Xinje XCPPro project, PLC1: XC3-32 (software 3.3q 2016-08-30)

PROGRAM Ladder

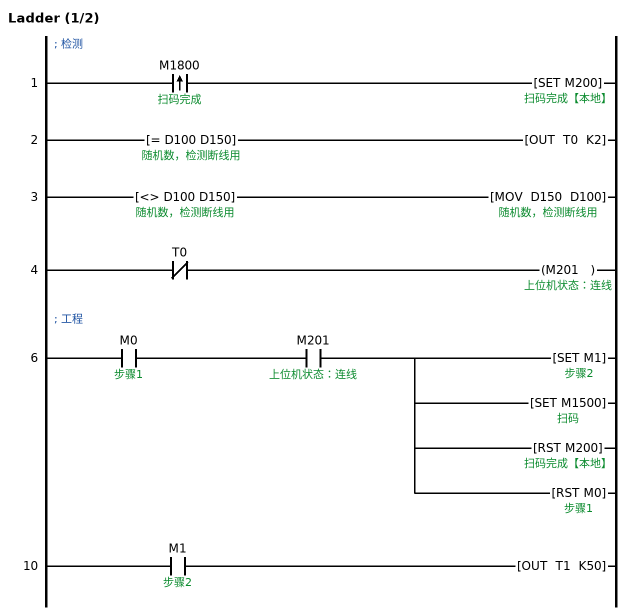
; 检测
LDP    M1800	; 扫码完成
SET    M200	; 扫码完成【本地】
LD=    D100 D150	; 随机数，检测断线用
OUT    T0 K2
LD<>   D100 D150	; 随机数，检测断线用
MOV    D150 D100	; 随机数，检测断线用
LDI    T0
OUT    M201	; 上位机状态：连线
; 工程
LD     M0	; 步骤1
AND    M201	; 上位机状态：连线
SET    M1	; 步骤2
SET    M1500	; 扫码
RST    M200	; 扫码完成【本地】
RST    M0	; 步骤1
LD     M1	; 步骤2
OUT    T1 K50

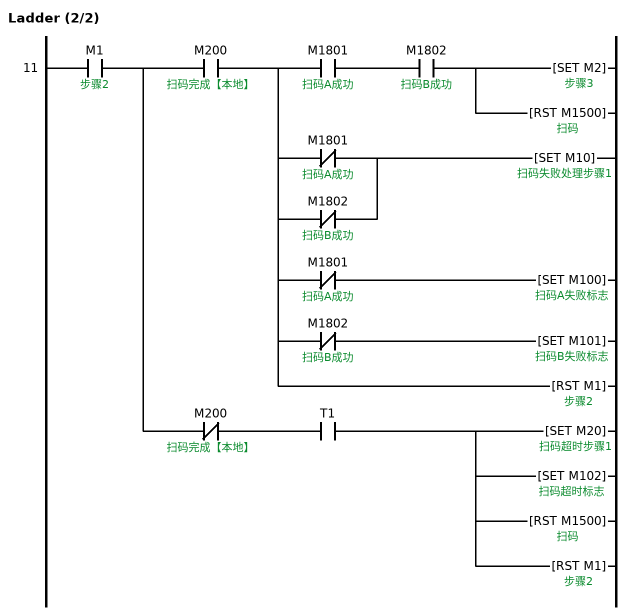
LD     M1	; 步骤2
MPS
AND    M200	; 扫码完成【本地】
MPS
AND    M1801	; 扫码A成功
AND    M1802	; 扫码B成功
SET    M2	; 步骤3
RST    M1500	; 扫码
MRD
LDI    M1801	; 扫码A成功
ORI    M1802	; 扫码B成功
ANB
SET    M10	; 扫码失败处理步骤1
MRD
ANI    M1801	; 扫码A成功
SET    M100	; 扫码A失败标志
MRD
ANI    M1802	; 扫码B成功
SET    M101	; 扫码B失败标志
MPP
RST    M1	; 步骤2
MPP
ANI    M200	; 扫码完成【本地】
AND    T1
SET    M20	; 扫码超时步骤1
SET    M102	; 扫码超时标志
RST    M1500	; 扫码
RST    M1	; 步骤2